TYPE st_AutoSperate :
STRUCT
Clips  		: ARRAY[0..4] OF BOOL; // Working Clips this round
Position 	: INT;				   // Position index 0~7
Row 		: INT;				   // Row of Needle 0~4
HandShake	: st_HandshakeBase;	   // Handshake
END_STRUCT
END_TYPE

(* stored: Version 1.1.0.1, ProductVersion 3.1.4024.13
   DUT st_AutoSperate: Id {686c74c3-e574-4592-a446-0ac9de204b2e} *)
